// This function has been automatically generated from the project information.
{attribute 'signature_flag' := '1073741824'}
{attribute 'TcGenerated'}
{attribute 'no-analysis'}
FUNCTION F_GetCompany : WSTRING
VAR_INPUT
	
END_VAR

F_GetCompany := "FisoThemes";

END_FUNCTION

(* stored: Version 1.1.0.1
   POU F_GetCompany: Id {e168c69e-69ad-4cd8-b6b7-1fe248ed7e37}, SpecialFunc None *)
